(*
Here we describe a function block, including some children.
*)
FUNCTION_BLOCK FB_ExampleFunctionBlock
VAR_INPUT
    input       : BOOL;
END_VAR
VAR_OUTPUT
    output      : STRING(15);
END_VAR

(*
Child method of our FB.
*)
METHOD ExampleMethod
VAR_INPUT
END_VAR
END_METHOD

(*
Reference to a variable that might be read-only.
*)
PROPERTY ExampleProperty : REFERENCE TO LREAL
GET
END_GET
SET
END_SET
END_PROPERTY

END_FUNCTION_BLOCK

(* stored: Version 1.1.0.1, ProductVersion 3.1.4024.11
   POU FB_ExampleFunctionBlock: Id {1d0f4647-a00a-42ef-8676-21cd880f317c}, SpecialFunc None
   Method ExampleMethod: Id {82381e22-448a-47e8-b264-9b857f411a3f}
   Property ExampleProperty: Id {cdcba121-a220-4eb8-8f4d-8924b3a02f60}
   Get Get: Id {fe3cd6e4-aa00-4539-98af-b9fb9586655f}
   Set Set: Id {80addca4-0610-47c4-8a76-38191658e0bd} *)
